FUNCTION_BLOCK DummyRollgang (* Template for a Basic Function Block Type *)
  (* Standard: 61499-2 *)
  (* Version 1.0, 2022-12-14, anubis *)
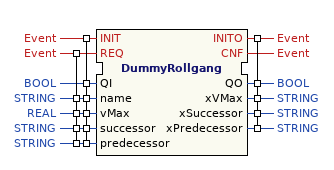
  EVENT_INPUT
    INIT WITH QI, name, vMax, successor, predecessor; (* Initialization Request *)
    REQ WITH name, vMax, successor, predecessor; (* Normal Execution Request *)
  END_EVENT
  EVENT_OUTPUT
    INITO WITH QO, xVMax, xSuccessor, xPredecessor; (* Initialization Confirm *)
    CNF; (* Execution Confirmation *)
  END_EVENT
  VAR_INPUT
    QI : BOOL; (* Input event qualifier *)
    name : STRING;
    vMax : REAL;
    successor : STRING;
    predecessor : STRING;
  END_VAR
  VAR_OUTPUT
    QO : BOOL; (* Output event qualifier *)
    xVMax : STRING;
    xSuccessor : STRING;
    xPredecessor : STRING;
  END_VAR
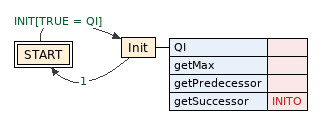
  EC_STATES
    START; (* Initial State *)
    Init : QI, getMax, getPredecessor, getSuccessor -> INITO; (* Initialization *)
  END_STATES
  EC_TRANSITIONS
    START TO Init := INIT[TRUE = QI];
    Init TO START := 1;
  END_TRANSITIONS
  ALGORITHM QI IN ST:
QO := QI;
  END_ALGORITHM
  ALGORITHM getMax IN ST:
xVMax := CONCAT('xquery ', STRING#'let $$name := $'', name, STRING#'$' ',
	'let $$component := //InstanceHierarchy/*/InternalElement[@Name=$$name] ',
	'let $$compType := tokenize($$component/RoleRequirements/@RefBaseRoleClassPath/data(),$'/$')[last()] ',
	'let $$rollerTable :=  $$component/InternalElement/RoleRequirements[contains(@RefBaseRoleClassPath,$'RollConveyor$')]/.. ',
	'let $$rollDiameter := $$rollerTable/Attribute[@Name=$'RollDiameter$']/Value/data() ',
	'let $$link := tokenize($$component/InternalLink/@RefPartnerSideA/data(),$':$')[1] ',
	'let $$motor := //InternalElement[@ID=$$link]/RoleRequirements[contains(@RefBaseRoleClassPath,$'ElectricMotor$')]/.. ',
	'let $$gearFactor := $$motor/Attribute[@Name=$'Gearfactor$']/Value/data() ',
	'let $$rotSpeed := $$motor/Attribute[@Name=$'Rotational Speed$']/Value/data() ',
	STRING#'let $$linSpeed :=  $$rotSpeed div (60.0 * $$gearFactor) * (2.0 * 3.1416 * 0.5 * $$rollDiameter) ',
	STRING#'return round-half-to-even($$linSpeed, 3)');
  END_ALGORITHM
  ALGORITHM getPredecessor IN ST:
xPredecessor := CONCAT(STRING#'xquery ', STRING#'let $$name := $'', name, STRING#'$' ',
	STRING#'let $$links := //InstanceHierarchy/InternalElement/InternalLink ',
	STRING#'let $$cp := //InstanceHierarchy/*/InternalElement[@Name=$$name] ', STRING#'let $$id := $$cp/@ID/data() ',
	STRING#'let $$succId := tokenize($$links[contains(@RefPartnerSideB, $$id)]/@RefPartnerSideA, $':$')[1] ',
	STRING#'let $$successor := //InstanceHierarchy/*/InternalElement[@ID=$$succId] ',
	STRING# 'return $$successor/@Name/data() ');
  END_ALGORITHM
  ALGORITHM getSuccessor IN ST:
xSuccessor := CONCAT('xquery ', STRING#'let $$name := $'', name, STRING#'$' ',
	STRING#'let $$links := //InstanceHierarchy/InternalElement/InternalLink ',
	STRING#'let $$cp := //InstanceHierarchy/*/InternalElement[@Name=$$name] ', STRING#'let $$id := $$cp/@ID/data() ',
	STRING#'let $$succId := tokenize($$links[contains(@RefPartnerSideA, $$id)]/@RefPartnerSideB, $':$')[1] ',
	STRING#'let $$successor := //InstanceHierarchy/*/InternalElement[@ID=$$succId] ',
	STRING# 'return $$successor/@Name/data() ');
  END_ALGORITHM
END_FUNCTION_BLOCK
